TYPE STATE:
    STRUCT
        curTime: LREAL;
        dvar_M_a: DINT;
    END_STRUCT;
END_TYPE
